FUNCTION_BLOCK E_STOPWATCH (* FB for stopping time between events *)
  PACKAGE eclipse4diac::utils::timing;
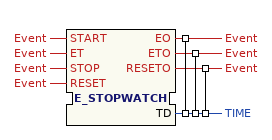
  EVENT_INPUT
    START; (* Start the stopwatch *)
    ET; (* Trigger the Time output *)
    STOP; (* Stop the stopwatch *)
    RESET; (* Reset the stopwatch to 0 *)
  END_EVENT
  EVENT_OUTPUT
    EO WITH TD; (* Event Output *)
    ETO WITH TD; (* Trigger the Time output  confirm *)
    RESETO WITH TD; (* Reset the stopwatch to 0  confirm *)
  END_EVENT
  VAR_OUTPUT
    TD : TIME; (* The measured time difference in milliseconds *)
  END_VAR
  VAR
    startTime : TIME; (* Holds the time value when the start event occured. *)
  END_VAR
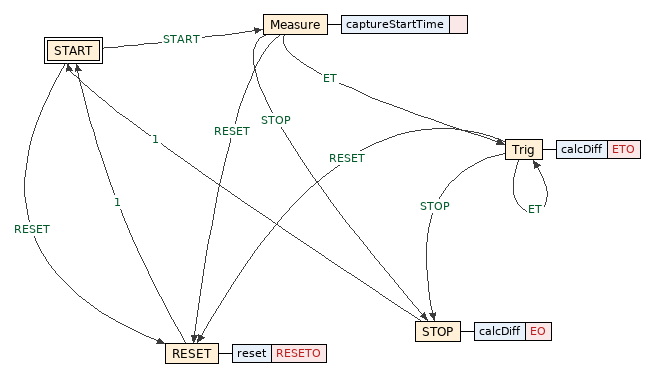
  EC_STATES
    START;
    Measure : captureStartTime;
    STOP : calcDiff -> EO;
    Trig : calcDiff -> ETO;
    RESET : reset -> RESETO;
  END_STATES
  EC_TRANSITIONS
    START TO Measure := START;
    Measure TO STOP := STOP;
    STOP TO START := 1;
    Trig TO STOP := STOP;
    Measure TO Trig := ET;
    Trig TO Trig := ET;
    Measure TO RESET := RESET;
    RESET TO START := 1;
    START TO RESET := RESET;
    Trig TO RESET := RESET;
  END_TRANSITIONS
  ALGORITHM captureStartTime IN ST:
startTime := NOW_MONOTONIC();
  END_ALGORITHM
  ALGORITHM calcDiff IN ST:
TD := NOW_MONOTONIC() - startTime;
  END_ALGORITHM
  ALGORITHM reset IN ST:
TD := T#0s;
  END_ALGORITHM
END_FUNCTION_BLOCK
